// TIA Portal V18 export
TYPE "udt_StoreRow"
// stored: IsFailsafeCompliant false
   STRUCT
      places : Array[0..5] of Bool;
   END_STRUCT;
END_TYPE
